SUBAPPLICATION Uebung_053_AX (* DigitalInput_I1-_I4 auf DigitalOutput_Q1-_Q4 *)
  (* Standard: 61499-2; Description: Copyright (c) 2023 Meisterschulen am Ostbahnhof This program and the accompanying materials are made available under the terms of the Eclipse Public License 2.0 which is available at https://www.eclipse.org/legal/epl-2.0/ SPDX-License-Identifier: EPL-2.0 *)
  (* Version 1.0, 2023-10-23, Franz Höpfinger, Meisterschulen am Ostbahnhof, initial API and implementation and/or initial documentation *)
  PACKAGE Uebungen;
  IMPORT logiBUS::io::DI::logiBUS_DI::Input_I1;
  IMPORT logiBUS::io::DI::logiBUS_DI::Input_I2;
  IMPORT logiBUS::io::DI::logiBUS_DI::Input_I3;
  IMPORT logiBUS::io::DI::logiBUS_DI::Input_I4;
  IMPORT logiBUS::io::DQ::logiBUS_DO::Output_Q1;
  IMPORT logiBUS::io::DQ::logiBUS_DO::Output_Q2;
  IMPORT logiBUS::io::DQ::logiBUS_DO::Output_Q3;
  IMPORT logiBUS::io::DQ::logiBUS_DO::Output_Q4;
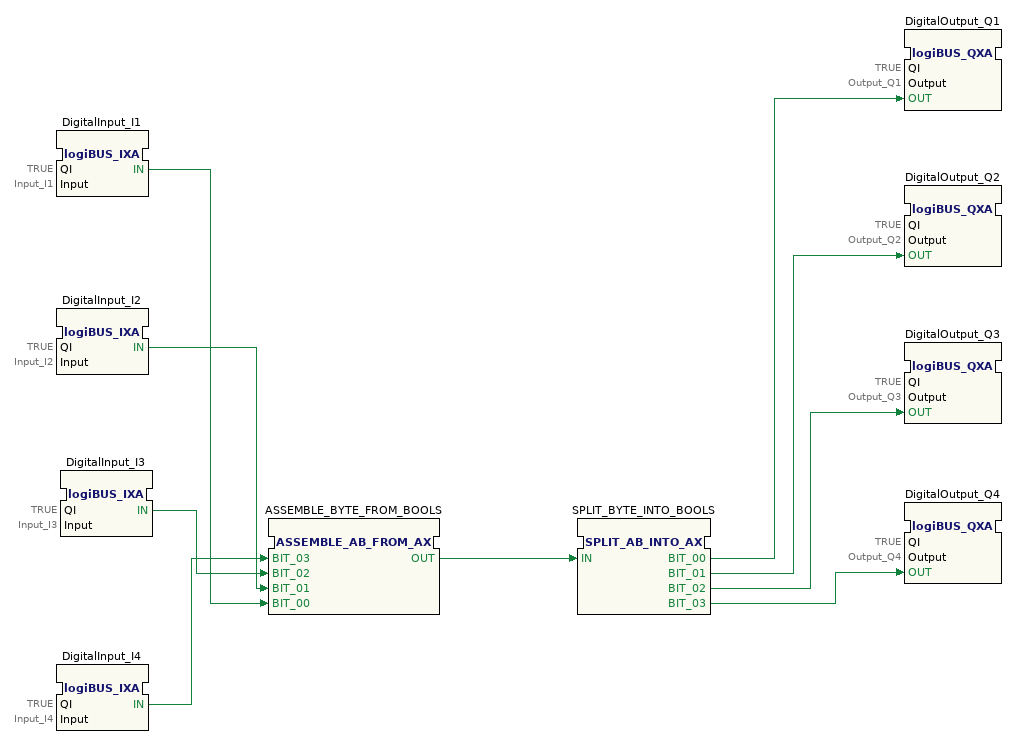
  FBS
    DigitalOutput_Q1 : logiBUS::io::DQ::logiBUS_QXA(QI := TRUE, Output := Output_Q1);
    DigitalInput_I1 : logiBUS::io::DI::logiBUS_IXA(QI := TRUE, Input := Input_I1);
    DigitalOutput_Q2 : logiBUS::io::DQ::logiBUS_QXA(QI := TRUE, Output := Output_Q2);
    DigitalInput_I2 : logiBUS::io::DI::logiBUS_IXA(QI := TRUE, Input := Input_I2);
    DigitalOutput_Q3 : logiBUS::io::DQ::logiBUS_QXA(QI := TRUE, Output := Output_Q3);
    DigitalInput_I3 : logiBUS::io::DI::logiBUS_IXA(QI := TRUE, Input := Input_I3);
    DigitalOutput_Q4 : logiBUS::io::DQ::logiBUS_QXA(QI := TRUE, Output := Output_Q4);
    DigitalInput_I4 : logiBUS::io::DI::logiBUS_IXA(QI := TRUE, Input := Input_I4);
    ASSEMBLE_BYTE_FROM_BOOLS : adapter::assembling::ASSEMBLE_AB_FROM_AX;
    SPLIT_BYTE_INTO_BOOLS : adapter::splitting::SPLIT_AB_INTO_AX;
  END_FBS
  ADAPTER_CONNECTIONS
    ASSEMBLE_BYTE_FROM_BOOLS.OUT TO SPLIT_BYTE_INTO_BOOLS.IN;
    SPLIT_BYTE_INTO_BOOLS.BIT_00 TO DigitalOutput_Q1.OUT;
    SPLIT_BYTE_INTO_BOOLS.BIT_01 TO DigitalOutput_Q2.OUT;
    SPLIT_BYTE_INTO_BOOLS.BIT_02 TO DigitalOutput_Q3.OUT;
    SPLIT_BYTE_INTO_BOOLS.BIT_03 TO DigitalOutput_Q4.OUT;
    DigitalInput_I4.IN TO ASSEMBLE_BYTE_FROM_BOOLS.BIT_03;
    DigitalInput_I3.IN TO ASSEMBLE_BYTE_FROM_BOOLS.BIT_02;
    DigitalInput_I2.IN TO ASSEMBLE_BYTE_FROM_BOOLS.BIT_01;
    DigitalInput_I1.IN TO ASSEMBLE_BYTE_FROM_BOOLS.BIT_00;
  END_CONNECTIONS
END_SUBAPPLICATION
